% RSLogix 500 project 8-31_BAK038.RSS, saved by version 8.10.00.18 %
PROJECT "UNTITLED"    % processor: MicroLogix 1400 %

PROGRAM FILES
  LAD 2   20 rungs

DATA FILES
  O0 OUTPUT  6 elements
  I1 INPUT  8 elements
  S2 STATUS  66 elements
  B3 BINARY  2 elements
  T4 TIMER  4 elements
  C5 COUNTER  1 elements
  R6 CONTROL  1 elements
  N7 INTEGER  1 elements
  F8 FLOAT  1 elements

LADDER 2
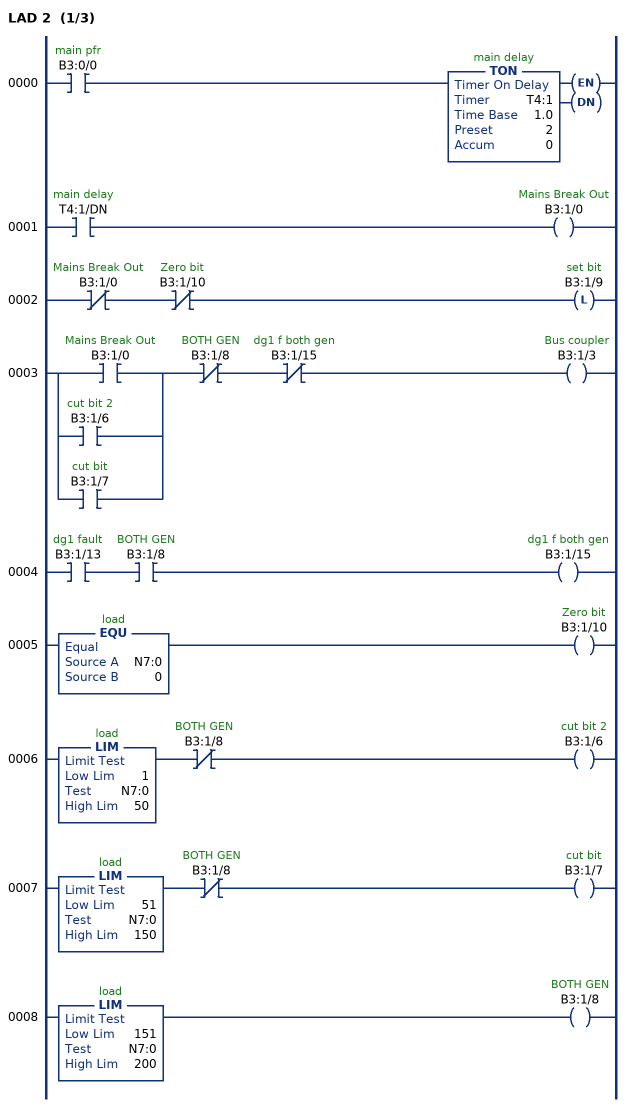
% Rung: 0 %
SOR XIC B3:0/0 TON T4:1 1.0 2 0 EOR
%   B3:0/0  "main pfr" %
%   T4:1  "main delay" %
% Rung: 1 %
SOR XIC T4:1/DN OTE B3:1/0 EOR
%   T4:1  "main delay" %
%   B3:1/0  "Mains Break Out" %
% Rung: 2 %
SOR XIO B3:1/0 XIO B3:1/10 OTL B3:1/9 EOR
%   B3:1/0  "Mains Break Out" %
%   B3:1/10  "Zero bit" %
%   B3:1/9  "set bit" %
% Rung: 3 %
SOR BST XIC B3:1/0 NXB BST XIC B3:1/6 NXB XIC B3:1/7 BND BND XIO B3:1/8 XIO B3:1/15 OTE B3:1/3 EOR
%   B3:1/0  "Mains Break Out" %
%   B3:1/6  "cut bit 2" %
%   B3:1/7  "cut bit" %
%   B3:1/8  "BOTH GEN" %
%   B3:1/15  "dg1 f both gen" %
%   B3:1/3  "Bus coupler" %
% Rung: 4 %
SOR XIC B3:1/13 XIC B3:1/8 OTE B3:1/15 EOR
%   B3:1/13  "dg1 fault" %
%   B3:1/8  "BOTH GEN" %
%   B3:1/15  "dg1 f both gen" %
% Rung: 5 %
SOR EQU N7:0 0 OTE B3:1/10 EOR
%   N7:0  "load" %
%   B3:1/10  "Zero bit" %
% Rung: 6 %
SOR LIM 1 N7:0 50 XIO B3:1/8 OTE B3:1/6 EOR
%   N7:0  "load" %
%   B3:1/8  "BOTH GEN" %
%   B3:1/6  "cut bit 2" %
% Rung: 7 %
SOR LIM 51 N7:0 150 XIO B3:1/8 OTE B3:1/7 EOR
%   N7:0  "load" %
%   B3:1/8  "BOTH GEN" %
%   B3:1/7  "cut bit" %
% Rung: 8 %
SOR LIM 151 N7:0 200 OTE B3:1/8 EOR
%   N7:0  "load" %
%   B3:1/8  "BOTH GEN" %

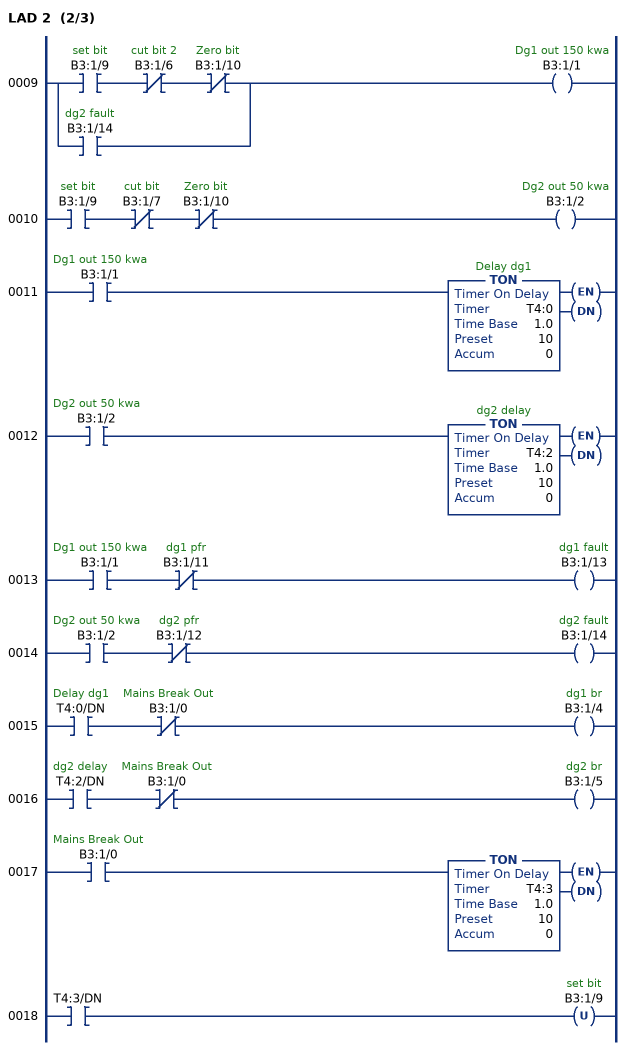
% Rung: 9 %
SOR BST XIC B3:1/9 XIO B3:1/6 XIO B3:1/10 NXB XIC B3:1/14 BND OTE B3:1/1 EOR
%   B3:1/9  "set bit" %
%   B3:1/6  "cut bit 2" %
%   B3:1/10  "Zero bit" %
%   B3:1/14  "dg2 fault" %
%   B3:1/1  "Dg1 out 150 kwa" %
% Rung: 10 %
SOR XIC B3:1/9 XIO B3:1/7 XIO B3:1/10 OTE B3:1/2 EOR
%   B3:1/9  "set bit" %
%   B3:1/7  "cut bit" %
%   B3:1/10  "Zero bit" %
%   B3:1/2  "Dg2 out 50 kwa" %
% Rung: 11 %
SOR XIC B3:1/1 TON T4:0 1.0 10 0 EOR
%   B3:1/1  "Dg1 out 150 kwa" %
%   T4:0  "Delay dg1" %
% Rung: 12 %
SOR XIC B3:1/2 TON T4:2 1.0 10 0 EOR
%   B3:1/2  "Dg2 out 50 kwa" %
%   T4:2  "dg2 delay" %
% Rung: 13 %
SOR XIC B3:1/1 XIO B3:1/11 OTE B3:1/13 EOR
%   B3:1/1  "Dg1 out 150 kwa" %
%   B3:1/11  "dg1 pfr" %
%   B3:1/13  "dg1 fault" %
% Rung: 14 %
SOR XIC B3:1/2 XIO B3:1/12 OTE B3:1/14 EOR
%   B3:1/2  "Dg2 out 50 kwa" %
%   B3:1/12  "dg2 pfr" %
%   B3:1/14  "dg2 fault" %
% Rung: 15 %
SOR XIC T4:0/DN XIO B3:1/0 OTE B3:1/4 EOR
%   T4:0  "Delay dg1" %
%   B3:1/0  "Mains Break Out" %
%   B3:1/4  "dg1 br" %
% Rung: 16 %
SOR XIC T4:2/DN XIO B3:1/0 OTE B3:1/5 EOR
%   T4:2  "dg2 delay" %
%   B3:1/0  "Mains Break Out" %
%   B3:1/5  "dg2 br" %
% Rung: 17 %
SOR XIC B3:1/0 TON T4:3 1.0 10 0 EOR
%   B3:1/0  "Mains Break Out" %
% Rung: 18 %
SOR XIC T4:3/DN OTU B3:1/9 EOR
%   B3:1/9  "set bit" %

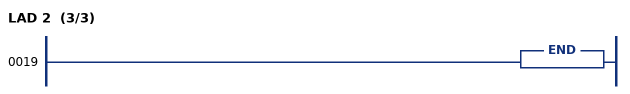
% Rung: 19 %
SOR END EOR

DATA TABLE (non-zero values as saved)
DATA B3
% B3:0 % 0X0000 0X029A
DATA T4
% .PRE .ACC %
% T4:0 % 10 0
% T4:1 % 2 0
% T4:2 % 10 0
% T4:3 % 10 0
